FUNCTION_BLOCK TLController (* Composite Function Block Type *)
  (* Standard: 61499-2 *)
  (* Version 0.2, 2003-12-05, JHC, Rockwell Automation, Renamed from NEWCOMPFB. *)
  (* Version 0.1, 2002-01-08, JHC, Rockwell Automation, Added DLY FB as example. *)
  (* Version 0.0, 2000-05-27, JHC, Rockwell Automation *)
  (* Compiler header: package fb.rt.template; *)
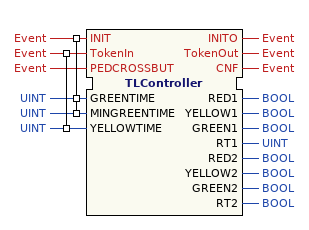
  EVENT_INPUT
    INIT WITH GREENTIME, MINGREENTIME; (* Initialization Request *)
    TokenIn WITH YELLOWTIME;
    PEDCROSSBUT;
  END_EVENT
  EVENT_OUTPUT
    INITO; (* Initialization Confirm *)
    TokenOut;
    CNF;
  END_EVENT
  VAR_INPUT
    GREENTIME : UINT;
    MINGREENTIME : UINT;
    YELLOWTIME : UINT;
  END_VAR
  VAR_OUTPUT
    RED1 : BOOL;
    YELLOW1 : BOOL;
    GREEN1 : BOOL;
    RT1 : UINT;
    RED2 : BOOL;
    YELLOW2 : BOOL;
    GREEN2 : BOOL;
    RT2 : BOOL;
  END_VAR
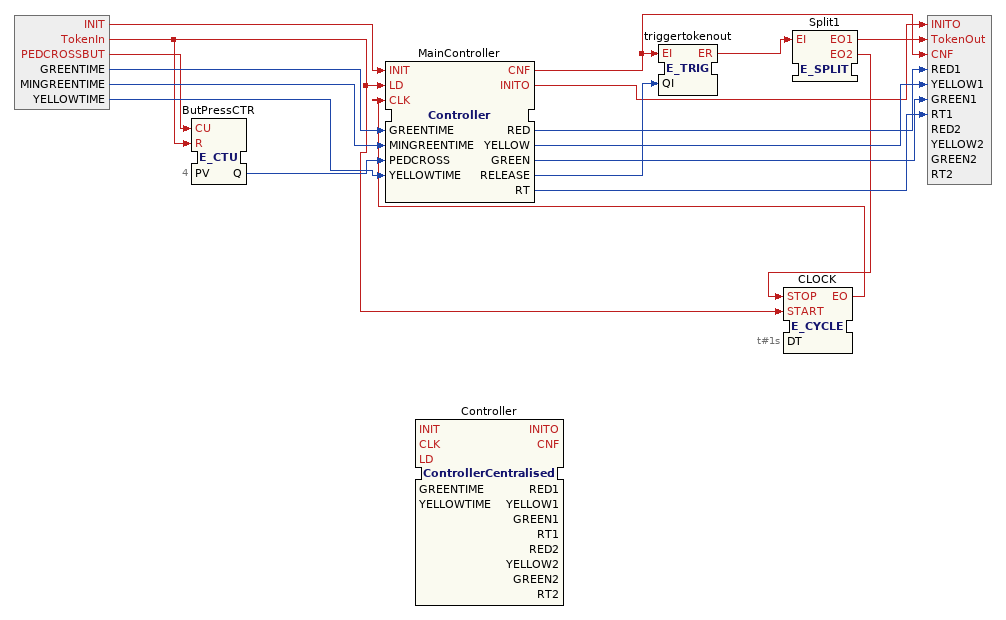
  FBS
    ButPressCTR : E_CTU(PV := 4);
    CLOCK : E_CYCLE(DT := t#1s);
    Split1 : E_SPLIT;
    triggertokenout : E_TRIG;
    MainController : Controller;
    Controller : ControllerCentralised;
  END_FBS
  EVENT_CONNECTIONS
    PEDCROSSBUT TO ButPressCTR.CU;
    Split1.EO1 TO TokenOut;
    Split1.EO2 TO CLOCK.STOP;
    triggertokenout.ER TO Split1.EI;
    TokenIn TO ButPressCTR.R;
    INIT TO MainController.INIT;
    TokenIn TO MainController.LD;
    MainController.CNF TO triggertokenout.EI;
    MainController.CNF TO CNF;
    MainController.INITO TO INITO;
    CLOCK.EO TO MainController.CLK;
    TokenIn TO CLOCK.START;
  END_CONNECTIONS
  DATA_CONNECTIONS
    GREENTIME TO MainController.GREENTIME;
    MINGREENTIME TO MainController.MINGREENTIME;
    ButPressCTR.Q TO MainController.PEDCROSS;
    YELLOWTIME TO MainController.YELLOWTIME;
    MainController.RED TO RED1;
    MainController.YELLOW TO YELLOW1;
    MainController.GREEN TO GREEN1;
    MainController.RELEASE TO triggertokenout.QI;
    MainController.RT TO RT1;
  END_CONNECTIONS
END_FUNCTION_BLOCK
